SUBAPPLICATION Ventilsteuerung (* Subapplication Type *)
  (* Standard: 61499-2 *)
  (* Version 1.0, 2023-10-23, franz *)
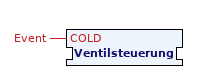
  EVENT_INPUT
    COLD;
  END_EVENT
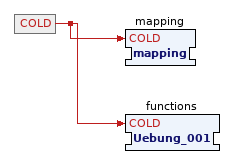
  SUBAPPS
    mapping : mapping;
    functions : Uebung_001;
  END_SUBAPPS
  EVENT_CONNECTIONS
    COLD TO mapping.COLD;
    COLD TO functions.COLD;
  END_CONNECTIONS
END_SUBAPPLICATION
